// TwinCAT 3 PLC project plc_sds_vis
// ProgramVersion: 3.1.4023.0
// libraries:
//   lcls-twincat-motion, * (SLAC)
//   Tc2_Standard, * (Beckhoff Automation GmbH)
//   Tc2_System, * (Beckhoff Automation GmbH)
//   Tc3_Module, * (Beckhoff Automation GmbH)
// project tree:
//   / PlcTask.TcTTO
//   POUs/ MAIN.TcPOU
// real-time tasks:
//   TASK PlcTask: cycle T#10ms, priority 20, ADS port 350
// motion (NC):
//   TASK NC-Task 1 SAF: cycle T#2ms, priority 4, ADS port 501
//   TASK NC-Task 1 SVB: cycle T#10ms, priority 8, ADS port 511
//   AXIS Axis 1 (id 1)
//   AXIS Axis 2 (id 2)
//   AXIS Axis 3 (id 3)
// I/O:
//   DEVICE Device 1 (EtherCAT), AmsNetId 172.21.148.78.2.1
//     Term 1 (EK1200) [EK1200-5000 EtherCAT Power supply (2A E-Bus)]
//       VIS-X (EL7037) [EL7037 1Ch. Stepper motor output stage (24V, 1.5A)]
//       VIS-Y (EL7037)
//       VIS-Z (EL7037)
//       Term 5 (EL9011)

CONFIGURATION plc_sds_vis
    RESOURCE PLC ON TwinCAT3
        TASK PlcTask(INTERVAL := T#10ms, PRIORITY := 20);
        PROGRAM MAIN WITH PlcTask : MAIN;
    END_RESOURCE
END_CONFIGURATION

// ---- POUs/MAIN.TcPOU
PROGRAM MAIN
VAR
     // Motor axes
    {attribute 'pytmc' := 'pv: VIS:MMS:X'}
    {attribute 'TcLinkTo' := '.bLimitForwardEnable  := TIID^Device 1 (EtherCAT)^Term 1 (EK1200)^VIS-X (EL7037)^STM Status^Status^Digital input 1;
                              .bLimitBackwardEnable := TIID^Device 1 (EtherCAT)^Term 1 (EK1200)^VIS-X (EL7037)^STM Status^Status^Digital input 2'}
    M1 : DUT_MotionStage := (bPowerSelf:=TRUE, nEnableMode:=ENUM_StageEnableMode.DURING_MOTION);
    fbVIS_X_Motor : FB_MotionStage;

    {attribute 'pytmc' := 'pv: VIS:MMS:Y'}
    {attribute 'TcLinkTo' := '.bLimitForwardEnable  := TIID^Device 1 (EtherCAT)^Term 1 (EK1200)^VIS-Y (EL7037)^STM Status^Status^Digital input 1;
                              .bLimitBackwardEnable := TIID^Device 1 (EtherCAT)^Term 1 (EK1200)^VIS-Y (EL7037)^STM Status^Status^Digital input 2'}
    M2 : DUT_MotionStage := (bPowerSelf:=TRUE, nEnableMode:=ENUM_StageEnableMode.DURING_MOTION);
    fbVIS_Y_Motor : FB_MotionStage;
    {attribute 'pytmc' := 'pv: VIS:MMS:Z'}
    {attribute 'TcLinkTo' := '.bLimitForwardEnable  := TIID^Device 1 (EtherCAT)^Term 1 (EK1200)^VIS-Z (EL7037)^STM Status^Status^Digital input 1;
                              .bLimitBackwardEnable := TIID^Device 1 (EtherCAT)^Term 1 (EK1200)^VIS-Z (EL7037)^STM Status^Status^Digital input 2'}
    M3 : DUT_MotionStage :=(bPowerSelf:=TRUE,nEnableMode:=ENUM_StageEnableMode.DURING_MOTION);
    fbVIS_Z_Motor : FB_MotionStage;
END_VAR

fbVIS_X_Motor(stMotionStage:=M1);
fbVIS_Y_Motor(stMotionStage:=M2);
fbVIS_Z_Motor(stMotionStage:=M3);

END_PROGRAM
